// LS Electric XG5000 project: T7_ETH_485_20221121_AfterHeat-CYB60-BT-AP4
// PLC NewPLC
// module base 0 slot 1: 내장위치결정:XBF-PO02E (오픈컬렉터형, 2축)
// module base 0 slot 2: Cnet:XBL-C41A (Cnet 통신 모듈(RS-422/485))

PROGRAM 7k_pwm (task: 스캔 프로그램)

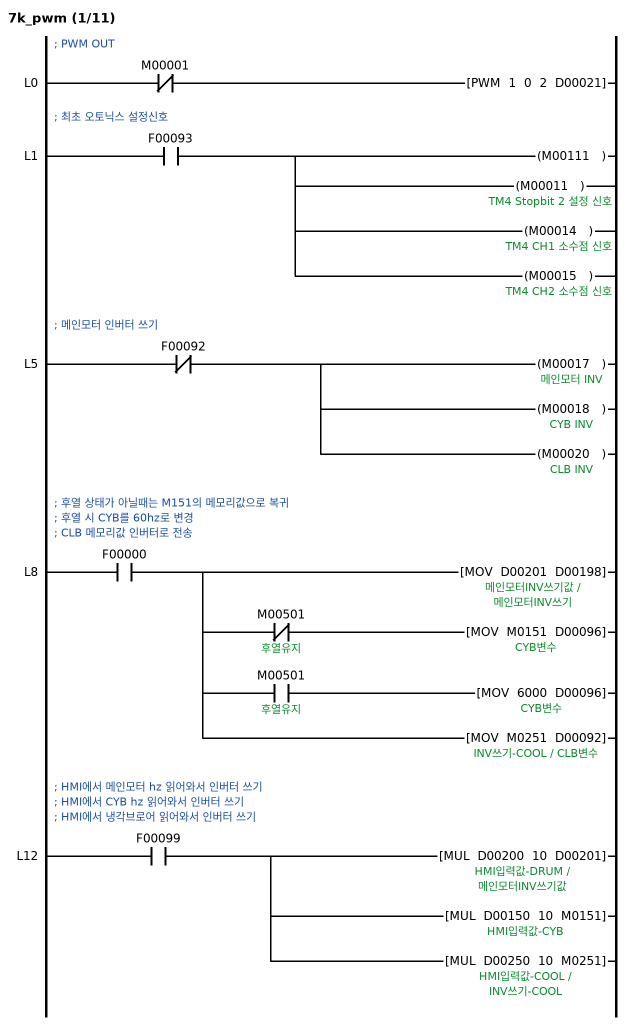
; L0
LOAD NOT  M00001
PWM       1 0 2 D00021
// output comment: PWM OUT
; L1
LOAD      F00093
OUT       M00111
OUT       M00011	// TM4 Stopbit 2 설정 신호
OUT       M00014	// TM4 CH1 소수점 신호
OUT       M00015	// TM4 CH2 소수점 신호
// output comment: 최초 오토닉스 설정신호
; L5
LOAD NOT  F00092
OUT       M00017	// 메인모터 INV
OUT       M00018	// CYB INV
OUT       M00020	// CLB INV
// output comment: 메인모터 인버터 쓰기
; L8
LOAD      F00000
MOV       D00201 D00198	// 메인모터INV쓰기값 / 메인모터INV쓰기
MPUSH
AND NOT   M00501	// 후열유지
MOV       M0151 D00096	// CYB변수
MLOAD
AND       M00501	// 후열유지
MOV       6000 D00096	// CYB변수
MPOP
MOV       M0251 D00092	// INV쓰기-COOL / CLB변수
// output comment: 후열 상태가 아닐때는 M151의 메모리값으로 복귀
// output comment: 후열 시 CYB를 60hz로 변경
// output comment: CLB 메모리값 인버터로 전송
; L12
LOAD      F00099
MUL       D00200 10 D00201	// HMI입력값-DRUM / 메인모터INV쓰기값
MUL       D00150 10 M0151	// HMI입력값-CYB
MUL       D00250 10 M0251	// HMI입력값-COOL / INV쓰기-COOL
// output comment: HMI에서 메인모터 hz 읽어와서 인버터 쓰기
// output comment: HMI에서 CYB hz 읽어와서 인버터 쓰기
// output comment: HMI에서 냉각브로어 읽어와서 인버터 쓰기

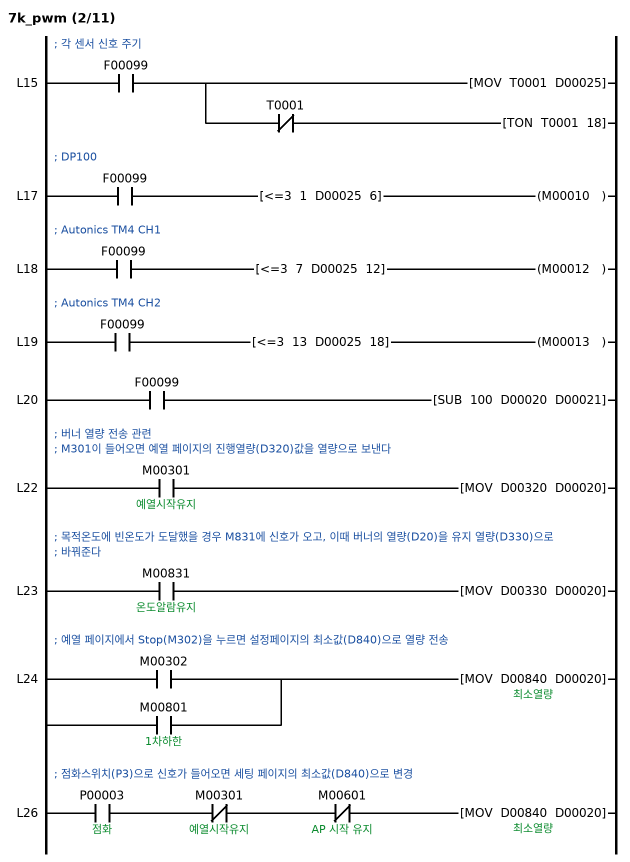
; L15
LOAD      F00099
MOV       T0001 D00025
AND NOT   T0001
TON       T0001 18
// output comment: 각 센서 신호 주기
; L17
LOAD      F00099
AND<=3    1 D00025 6
OUT       M00010
// output comment: DP100
; L18
LOAD      F00099
AND<=3    7 D00025 12
OUT       M00012
// output comment: Autonics TM4 CH1
; L19
LOAD      F00099
AND<=3    13 D00025 18
OUT       M00013
// output comment: Autonics TM4 CH2
; L20
LOAD      F00099
SUB       100 D00020 D00021
// 버너 열량 전송 관련
; L22
LOAD      M00301	// 예열시작유지
MOV       D00320 D00020
// output comment: M301이 들어오면 예열 페이지의 진행열량(D320)값을 열량으로 보낸다
; L23
LOAD      M00831	// 온도알람유지
MOV       D00330 D00020
// output comment: 목적온도에 빈온도가 도달했을 경우 M831에 신호가 오고, 이때 버너의 열량(D20)을 유지 열량(D330)으로 바꿔준다
; L24
LOAD      M00302
OR        M00801	// 1차하한
MOV       D00840 D00020	// 최소열량
// output comment: 예열 페이지에서 Stop(M302)을 누르면 설정페이지의 최소값(D840)으로 열량 전송
; L26
LOAD      P00003	// 점화
AND NOT   M00301	// 예열시작유지
AND NOT   M00601	// AP 시작 유지
MOV       D00840 D00020	// 최소열량
// output comment: 점화스위치(P3)으로 신호가 들어오면 세팅 페이지의 최소값(D840)으로 변경

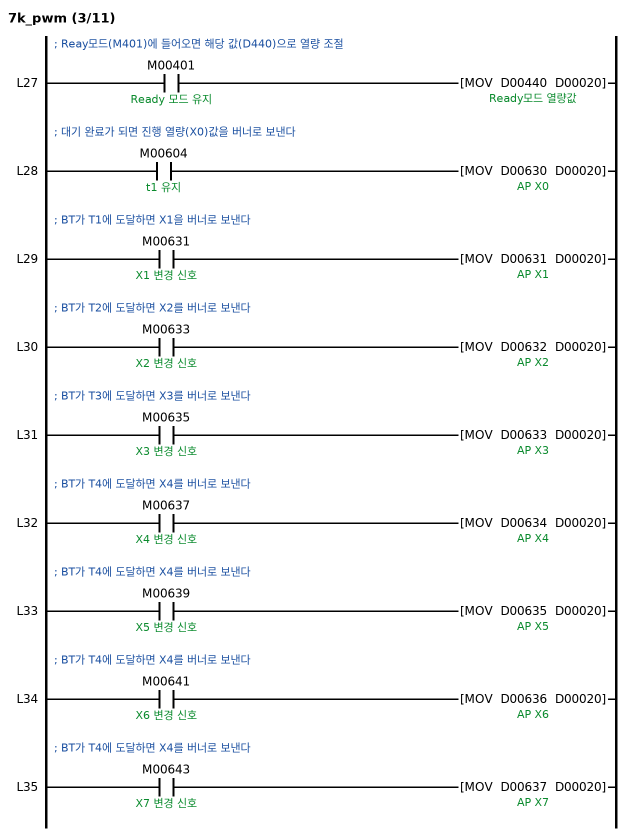
; L27
LOAD      M00401	// Ready 모드 유지
MOV       D00440 D00020	// Ready모드 열량값
// output comment: Reay모드(M401)에 들어오면 해당 값(D440)으로 열량 조절
; L28
LOAD      M00604	// t1 유지
MOV       D00630 D00020	// AP X0
// output comment: 대기 완료가 되면 진행 열량(X0)값을 버너로 보낸다
; L29
LOAD      M00631	// X1 변경 신호
MOV       D00631 D00020	// AP X1
// output comment: BT가 T1에 도달하면 X1을 버너로 보낸다
; L30
LOAD      M00633	// X2 변경 신호
MOV       D00632 D00020	// AP X2
// output comment: BT가 T2에 도달하면 X2를 버너로 보낸다
; L31
LOAD      M00635	// X3 변경 신호
MOV       D00633 D00020	// AP X3
// output comment: BT가 T3에 도달하면 X3를 버너로 보낸다
; L32
LOAD      M00637	// X4 변경 신호
MOV       D00634 D00020	// AP X4
// output comment: BT가 T4에 도달하면 X4를 버너로 보낸다
; L33
LOAD      M00639	// X5 변경 신호
MOV       D00635 D00020	// AP X5
// output comment: BT가 T4에 도달하면 X4를 버너로 보낸다
; L34
LOAD      M00641	// X6 변경 신호
MOV       D00636 D00020	// AP X6
// output comment: BT가 T4에 도달하면 X4를 버너로 보낸다
; L35
LOAD      M00643	// X7 변경 신호
MOV       D00637 D00020	// AP X7
// output comment: BT가 T4에 도달하면 X4를 버너로 보낸다

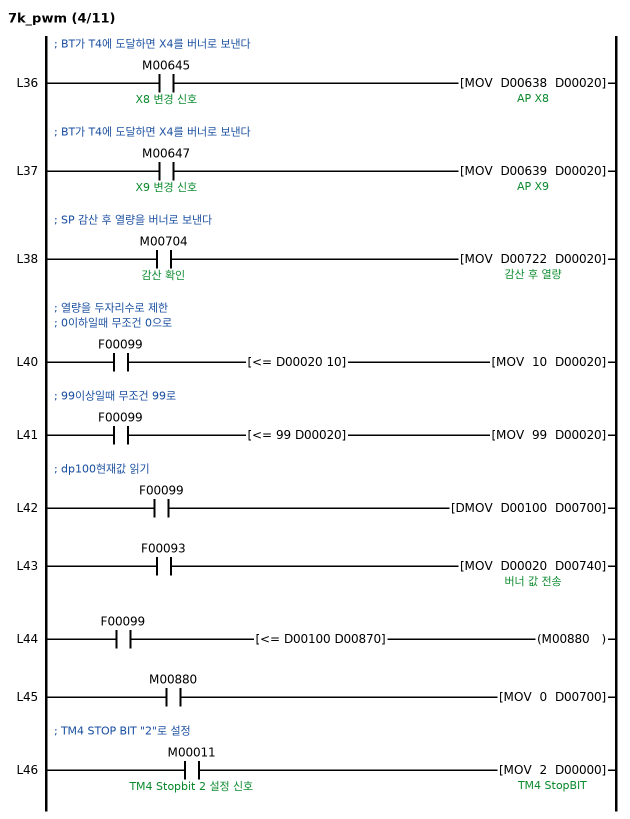
; L36
LOAD      M00645	// X8 변경 신호
MOV       D00638 D00020	// AP X8
// output comment: BT가 T4에 도달하면 X4를 버너로 보낸다
; L37
LOAD      M00647	// X9 변경 신호
MOV       D00639 D00020	// AP X9
// output comment: BT가 T4에 도달하면 X4를 버너로 보낸다
; L38
LOAD      M00704	// 감산 확인
MOV       D00722 D00020	// 감산 후 열량
// output comment: SP 감산 후 열량을 버너로 보낸다
// 열량을 두자리수로 제한
; L40
LOAD      F00099
AND<=     D00020 10
MOV       10 D00020
// output comment: 0이하일때 무조건 0으로
; L41
LOAD      F00099
AND<=     99 D00020
MOV       99 D00020
// output comment: 99이상일때 무조건 99로
; L42
LOAD      F00099
DMOV      D00100 D00700
// output comment: dp100현재값 읽기
; L43
LOAD      F00093
MOV       D00020 D00740	// 버너 값 전송
; L44
LOAD      F00099
AND<=     D00100 D00870
OUT       M00880
; L45
LOAD      M00880
MOV       0 D00700
; L46
LOAD      M00011	// TM4 Stopbit 2 설정 신호
MOV       2 D00000	// TM4 StopBIT
// output comment: TM4 STOP BIT "2"로 설정

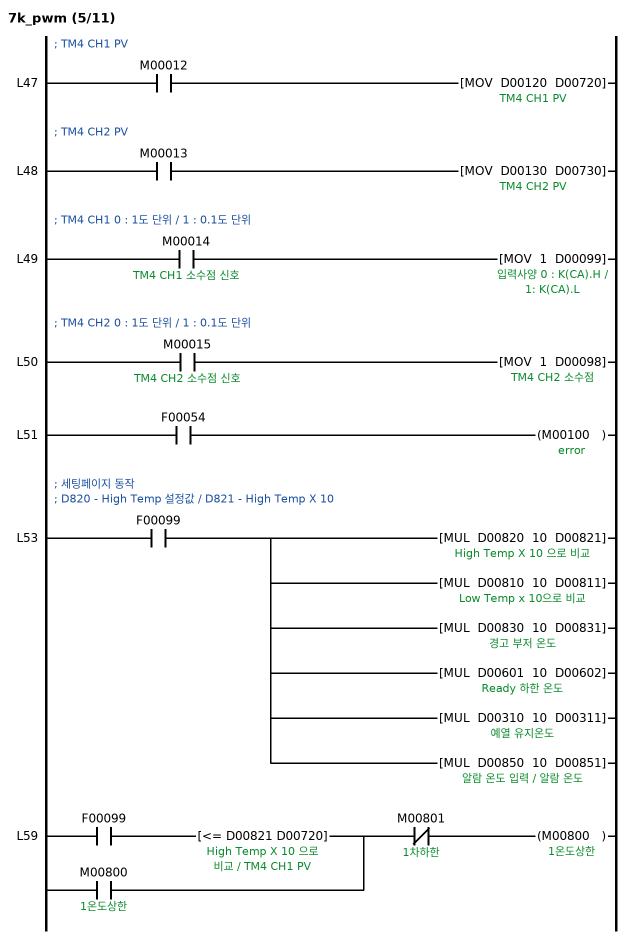
; L47
LOAD      M00012
MOV       D00120 D00720	// TM4 CH1 PV
// output comment: TM4 CH1 PV
; L48
LOAD      M00013
MOV       D00130 D00730	// TM4 CH2 PV
// output comment: TM4 CH2 PV
; L49
LOAD      M00014	// TM4 CH1 소수점 신호
MOV       1 D00099	// 입력사양 0 : K(CA).H / 1: K(CA).L
// output comment: TM4 CH1 0 : 1도 단위 / 1 : 0.1도 단위
; L50
LOAD      M00015	// TM4 CH2 소수점 신호
MOV       1 D00098	// TM4 CH2 소수점
// output comment: TM4 CH2 0 : 1도 단위 / 1 : 0.1도 단위
; L51
LOAD      F00054
OUT       M00100	// error
// 세팅페이지 동작
; L53
LOAD      F00099
MUL       D00820 10 D00821	// High Temp X 10 으로 비교
MUL       D00810 10 D00811	// Low Temp x 10으로 비교
MUL       D00830 10 D00831	// 경고 부저 온도
MUL       D00601 10 D00602	// Ready 하한 온도
MUL       D00310 10 D00311	// 예열 유지온도
MUL       D00850 10 D00851	// 알람 온도 입력 / 알람 온도 
// output comment: D820 - High Temp 설정값 / D821 - High Temp X 10
; L59
LOAD      F00099
AND<=     D00821 D00720	// High Temp X 10 으로 비교 / TM4 CH1 PV
OR        M00800	// 1온도상한
AND NOT   M00801	// 1차하한
OUT       M00800	// 1온도상한

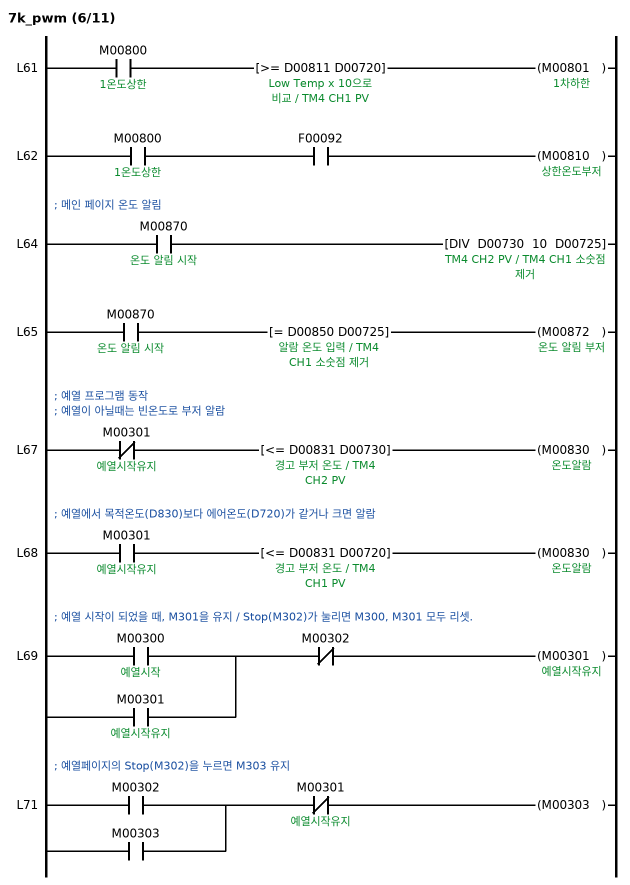
; L61
LOAD      M00800	// 1온도상한
AND>=     D00811 D00720	// Low Temp x 10으로 비교 / TM4 CH1 PV
OUT       M00801	// 1차하한
; L62
LOAD      M00800	// 1온도상한
AND       F00092
OUT       M00810	// 상한온도부저
// 메인 페이지 온도 알림
; L64
LOAD      M00870	// 온도 알림 시작
DIV       D00730 10 D00725	// TM4 CH2 PV / TM4 CH1 소숫점 제거
; L65
LOAD      M00870	// 온도 알림 시작
AND=      D00850 D00725	// 알람 온도 입력 / TM4 CH1 소숫점 제거
OUT       M00872	// 온도 알림 부저
// 예열 프로그램 동작
; L67
LOAD NOT  M00301	// 예열시작유지
AND<=     D00831 D00730	// 경고 부저 온도 / TM4 CH2 PV
OUT       M00830	// 온도알람
// output comment: 예열이 아닐때는 빈온도로 부저 알람
; L68
LOAD      M00301	// 예열시작유지
AND<=     D00831 D00720	// 경고 부저 온도 / TM4 CH1 PV
OUT       M00830	// 온도알람
// output comment: 예열에서 목적온도(D830)보다 에어온도(D720)가 같거나 크면 알람
; L69
LOAD      M00300	// 예열시작
OR        M00301	// 예열시작유지
AND NOT   M00302
OUT       M00301	// 예열시작유지
// output comment: 예열 시작이 되었을 때, M301을 유지 / Stop(M302)가 눌리면 M300, M301 모두 리셋.
; L71
LOAD      M00302
OR        M00303
AND NOT   M00301	// 예열시작유지
OUT       M00303
// output comment: 예열페이지의 Stop(M302)을 누르면 M303 유지

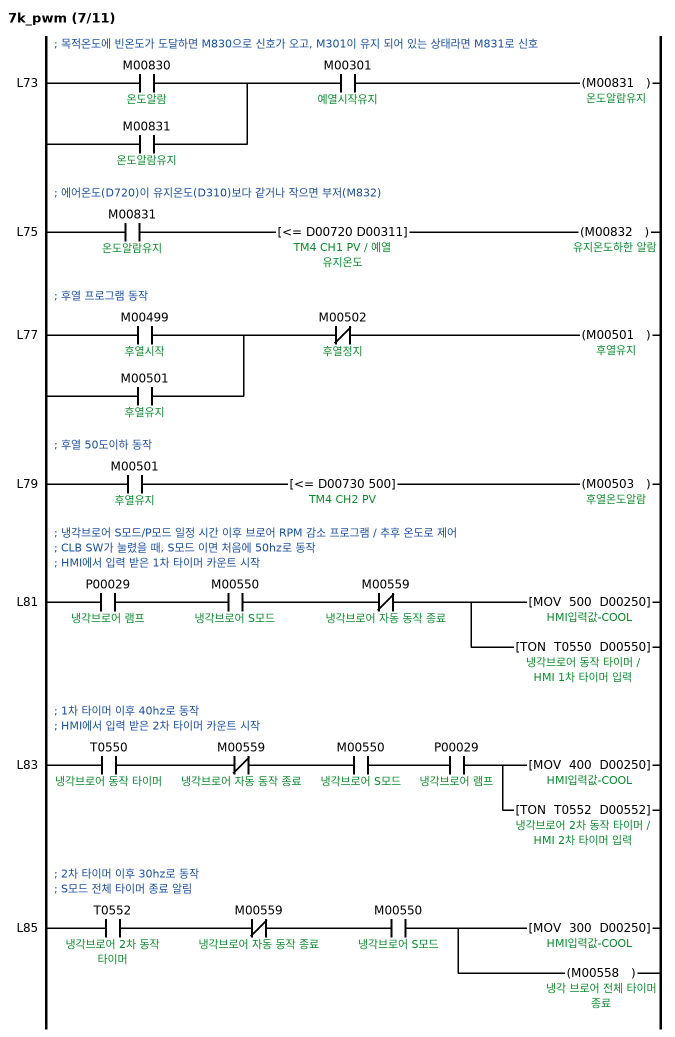
; L73
LOAD      M00830	// 온도알람
OR        M00831	// 온도알람유지
AND       M00301	// 예열시작유지
OUT       M00831	// 온도알람유지
// output comment: 목적온도에 빈온도가 도달하면 M830으로 신호가 오고, M301이 유지 되어 있는 상태라면 M831로 신호
; L75
LOAD      M00831	// 온도알람유지
AND<=     D00720 D00311	// TM4 CH1 PV / 예열 유지온도
OUT       M00832	// 유지온도하한 알람
// output comment: 에어온도(D720)이 유지온도(D310)보다 같거나 작으면 부저(M832)
// 후열 프로그램 동작
; L77
LOAD      M00499	// 후열시작
OR        M00501	// 후열유지
AND NOT   M00502	// 후열정지
OUT       M00501	// 후열유지
; L79
LOAD      M00501	// 후열유지
AND<=     D00730 500	// TM4 CH2 PV
OUT       M00503	// 후열온도알람
// output comment: 후열 50도이하 동작
// 냉각브로어 S모드/P모드 일정 시간 이후 브로어 RPM 감소 프로그램 / 추후 온도로 제어
; L81
LOAD      P00029	// 냉각브로어 램프
AND       M00550	// 냉각브로어 S모드
AND NOT   M00559	// 냉각브로어 자동 동작 종료
MOV       500 D00250	// HMI입력값-COOL
TON       T0550 D00550	// 냉각브로어 동작 타이머 / HMI 1차 타이머 입력
// output comment: CLB SW가 눌렸을 때, S모드 이면 처음에 50hz로 동작
// output comment: HMI에서 입력 받은 1차 타이머 카운트 시작
; L83
LOAD      T0550	// 냉각브로어 동작 타이머
AND NOT   M00559	// 냉각브로어 자동 동작 종료
AND       M00550	// 냉각브로어 S모드
AND       P00029	// 냉각브로어 램프
MOV       400 D00250	// HMI입력값-COOL
TON       T0552 D00552	// 냉각브로어 2차 동작 타이머 / HMI 2차 타이머 입력
// output comment: 1차 타이머 이후 40hz로 동작
// output comment: HMI에서 입력 받은 2차 타이머 카운트 시작
; L85
LOAD      T0552	// 냉각브로어 2차 동작 타이머
AND NOT   M00559	// 냉각브로어 자동 동작 종료
AND       M00550	// 냉각브로어 S모드
MOV       300 D00250	// HMI입력값-COOL
OUT       M00558	// 냉각 브로어 전체 타이머 종료
// output comment: 2차 타이머 이후 30hz로 동작
// output comment: S모드 전체 타이머 종료 알림

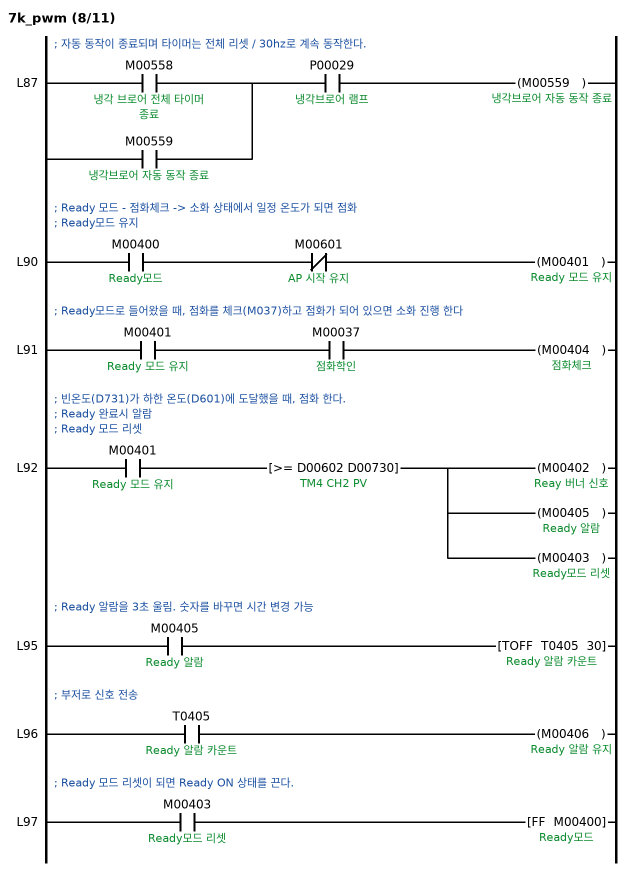
; L87
LOAD      M00558	// 냉각 브로어 전체 타이머 종료
OR        M00559	// 냉각브로어 자동 동작 종료
AND       P00029	// 냉각브로어 램프
OUT       M00559	// 냉각브로어 자동 동작 종료
// output comment: 자동 동작이 종료되며 타이머는 전체 리셋 / 30hz로 계속 동작한다.
// Ready 모드 - 점화체크 -> 소화 상태에서 일정 온도가 되면 점화
; L90
LOAD      M00400	// Ready모드
AND NOT   M00601	// AP 시작 유지
OUT       M00401	// Ready 모드 유지
// output comment: Ready모드 유지
; L91
LOAD      M00401	// Ready 모드 유지
AND       M00037	// 점화학인
OUT       M00404	// 점화체크
// output comment: Ready모드로 들어왔을 때, 점화를 체크(M037)하고 점화가 되어 있으면 소화 진행 한다
; L92
LOAD      M00401	// Ready 모드 유지
AND>=     D00602 D00730	// TM4 CH2 PV
OUT       M00402	// Reay 버너 신호
OUT       M00405	// Ready 알람
OUT       M00403	// Ready모드 리셋
// output comment: 빈온도(D731)가 하한 온도(D601)에 도달했을 때, 점화 한다.
// output comment: Ready 완료시 알람
// output comment: Ready 모드 리셋
; L95
LOAD      M00405	// Ready 알람
TOFF      T0405 30	// Ready 알람 카운트
// output comment: Ready 알람을 3초 울림. 숫자를 바꾸면 시간 변경 가능
; L96
LOAD      T0405	// Ready 알람 카운트
OUT       M00406	// Ready 알람 유지
// output comment: 부저로 신호 전송
; L97
LOAD      M00403	// Ready모드 리셋
FF        M00400	// Ready모드
// output comment: Ready 모드 리셋이 되면 Ready ON 상태를 끈다.

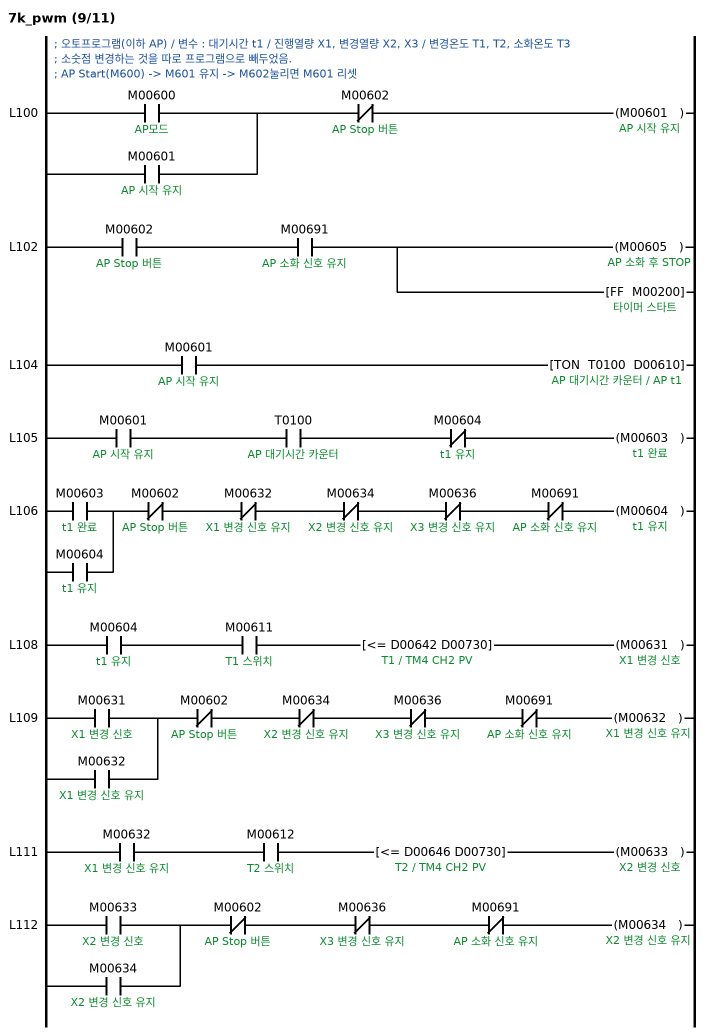
// 오토프로그램(이하 AP) / 변수 : 대기시간 t1 / 진행열량 X1, 변경열량 X2, X3 / 변경온도 T1, T2, 소화온도 T3
// 소숫점 변경하는 것을 따로 프로그램으로 빼두었음.
; L100
LOAD      M00600	// AP모드
OR        M00601	// AP 시작 유지
AND NOT   M00602	// AP Stop 버튼
OUT       M00601	// AP 시작 유지
// output comment: AP Start(M600) -> M601 유지 -> M602눌리면 M601 리셋
; L102
LOAD      M00602	// AP Stop 버튼
AND       M00691	// AP 소화 신호 유지
OUT       M00605	// AP 소화 후 STOP
FF        M00200	// 타이머 스타트
; L104
LOAD      M00601	// AP 시작 유지
TON       T0100 D00610	// AP 대기시간 카운터 / AP t1
; L105
LOAD      M00601	// AP 시작 유지
AND       T0100	// AP 대기시간 카운터
AND NOT   M00604	// t1 유지
OUT       M00603	// t1 완료
; L106
LOAD      M00603	// t1 완료
OR        M00604	// t1 유지
AND NOT   M00602	// AP Stop 버튼
AND NOT   M00632	// X1 변경 신호 유지
AND NOT   M00634	// X2 변경 신호 유지
AND NOT   M00636	// X3 변경 신호 유지
AND NOT   M00691	// AP 소화 신호 유지
OUT       M00604	// t1 유지
; L108
LOAD      M00604	// t1 유지
AND       M00611	// T1 스위치
AND<=     D00642 D00730	// T1 / TM4 CH2 PV
OUT       M00631	// X1 변경 신호
; L109
LOAD      M00631	// X1 변경 신호
OR        M00632	// X1 변경 신호 유지
AND NOT   M00602	// AP Stop 버튼
AND NOT   M00634	// X2 변경 신호 유지
AND NOT   M00636	// X3 변경 신호 유지
AND NOT   M00691	// AP 소화 신호 유지
OUT       M00632	// X1 변경 신호 유지
; L111
LOAD      M00632	// X1 변경 신호 유지
AND       M00612	// T2 스위치
AND<=     D00646 D00730	// T2 / TM4 CH2 PV
OUT       M00633	// X2 변경 신호
; L112
LOAD      M00633	// X2 변경 신호
OR        M00634	// X2 변경 신호 유지
AND NOT   M00602	// AP Stop 버튼
AND NOT   M00636	// X3 변경 신호 유지
AND NOT   M00691	// AP 소화 신호 유지
OUT       M00634	// X2 변경 신호 유지

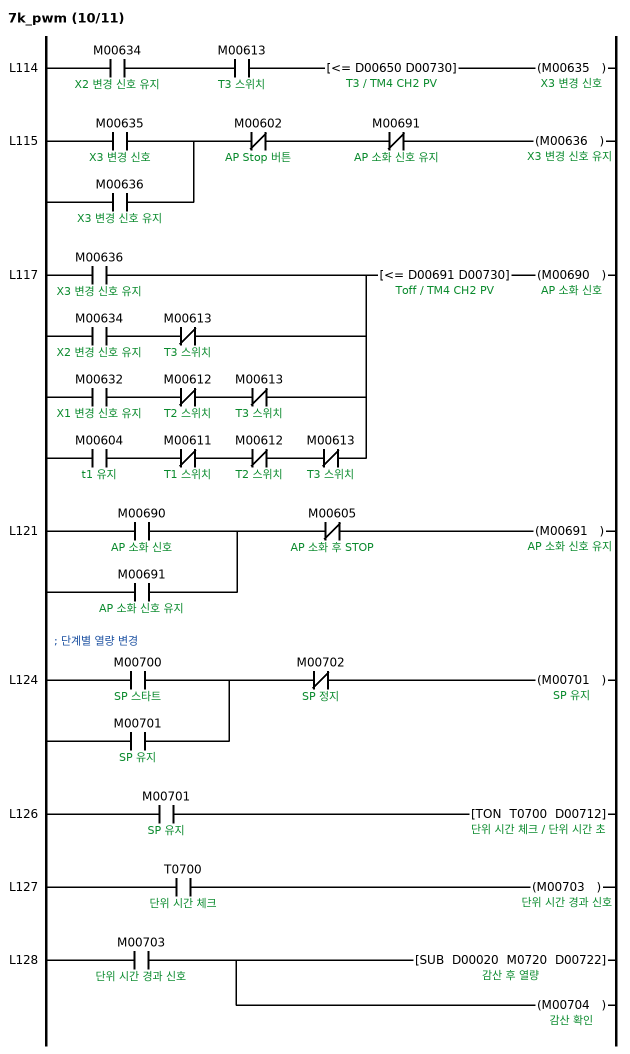
; L114
LOAD      M00634	// X2 변경 신호 유지
AND       M00613	// T3 스위치
AND<=     D00650 D00730	// T3 / TM4 CH2 PV
OUT       M00635	// X3 변경 신호
; L115
LOAD      M00635	// X3 변경 신호
OR        M00636	// X3 변경 신호 유지
AND NOT   M00602	// AP Stop 버튼
AND NOT   M00691	// AP 소화 신호 유지
OUT       M00636	// X3 변경 신호 유지
; L117
LOAD      M00636	// X3 변경 신호 유지
LOAD      M00634	// X2 변경 신호 유지
AND NOT   M00613	// T3 스위치
OR LOAD
LOAD      M00632	// X1 변경 신호 유지
AND NOT   M00612	// T2 스위치
AND NOT   M00613	// T3 스위치
OR LOAD
LOAD      M00604	// t1 유지
AND NOT   M00611	// T1 스위치
AND NOT   M00612	// T2 스위치
AND NOT   M00613	// T3 스위치
OR LOAD
AND<=     D00691 D00730	// Toff / TM4 CH2 PV
OUT       M00690	// AP 소화 신호
; L121
LOAD      M00690	// AP 소화 신호
OR        M00691	// AP 소화 신호 유지
AND NOT   M00605	// AP 소화 후 STOP
OUT       M00691	// AP 소화 신호 유지
// 단계별 열량 변경
; L124
LOAD      M00700	// SP 스타트
OR        M00701	// SP 유지
AND NOT   M00702	// SP 정지
OUT       M00701	// SP 유지
; L126
LOAD      M00701	// SP 유지
TON       T0700 D00712	// 단위 시간 체크 / 단위 시간 초
; L127
LOAD      T0700	// 단위 시간 체크
OUT       M00703	// 단위 시간 경과 신호
; L128
LOAD      M00703	// 단위 시간 경과 신호
SUB       D00020 M0720 D00722	// 감산 후 열량
OUT       M00704	// 감산 확인

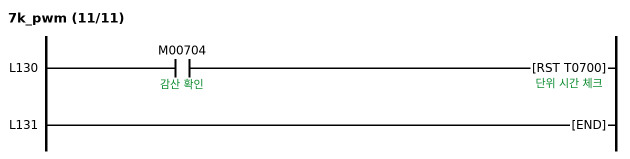
; L130
LOAD      M00704	// 감산 확인
RST       T0700	// 단위 시간 체크
; L131
END

PROGRAM 타이머 (task: 스캔 프로그램)

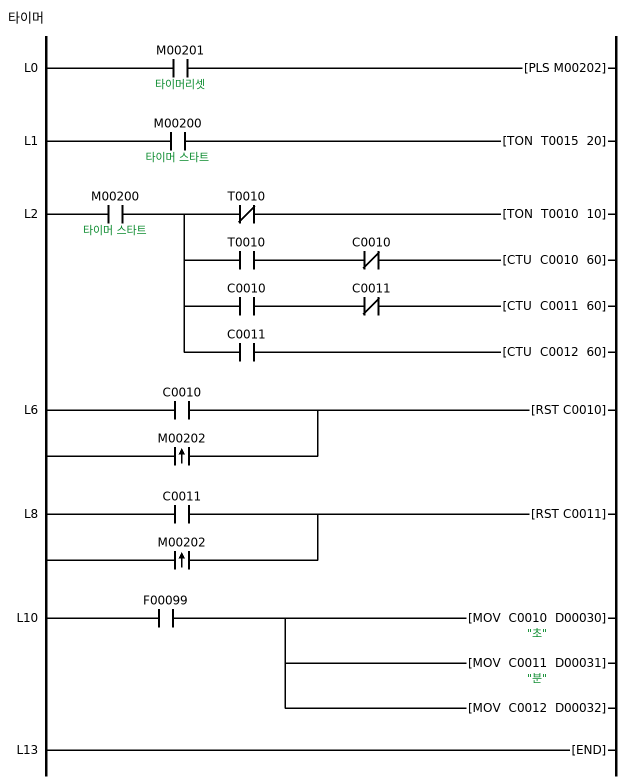
; L0
LOAD      M00201	// 타이머리셋
OUTP      M00202
; L1
LOAD      M00200	// 타이머 스타트
TON       T0015 20
; L2
LOAD      M00200	// 타이머 스타트
MPUSH
AND NOT   T0010
TON       T0010 10
MLOAD
AND       T0010
AND NOT   C0010
CTU       C0010 60
MLOAD
AND       C0010
AND NOT   C0011
CTU       C0011 60
MPOP
AND       C0011
CTU       C0012 60
; L6
LOAD      C0010
ORP       M00202
RST       C0010
; L8
LOAD      C0011
ORP       M00202
RST       C0011
; L10
LOAD      F00099
MOV       C0010 D00030	// "초"
MOV       C0011 D00031	// "분"
MOV       C0012 D00032
; L13
END

PROGRAM control (task: 스캔 프로그램)

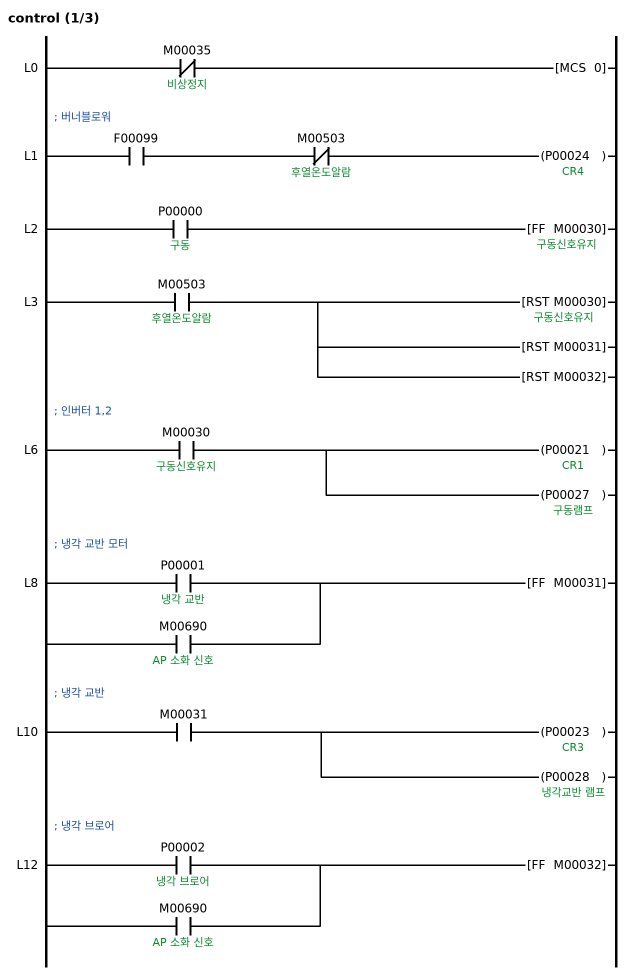
; L0
LOAD NOT  M00035	// 비상정지
MCS       0
; L1
LOAD      F00099
AND NOT   M00503	// 후열온도알람
OUT       P00024	// CR4
// output comment: 버너블로워
; L2
LOAD      P00000	// 구동
FF        M00030	// 구동신호유지
; L3
LOAD      M00503	// 후열온도알람
RST       M00030	// 구동신호유지
RST       M00031
RST       M00032
; L6
LOAD      M00030	// 구동신호유지
OUT       P00021	// CR1
OUT       P00027	// 구동램프
// output comment: 인버터 1,2
; L8
LOAD      P00001	// 냉각 교반
OR        M00690	// AP 소화 신호
FF        M00031
// output comment: 냉각 교반 모터
; L10
LOAD      M00031
OUT       P00023	// CR3
OUT       P00028	// 냉각교반 램프
// output comment: 냉각 교반
; L12
LOAD      P00002	// 냉각 브로어
OR        M00690	// AP 소화 신호
FF        M00032
// output comment: 냉각 브로어

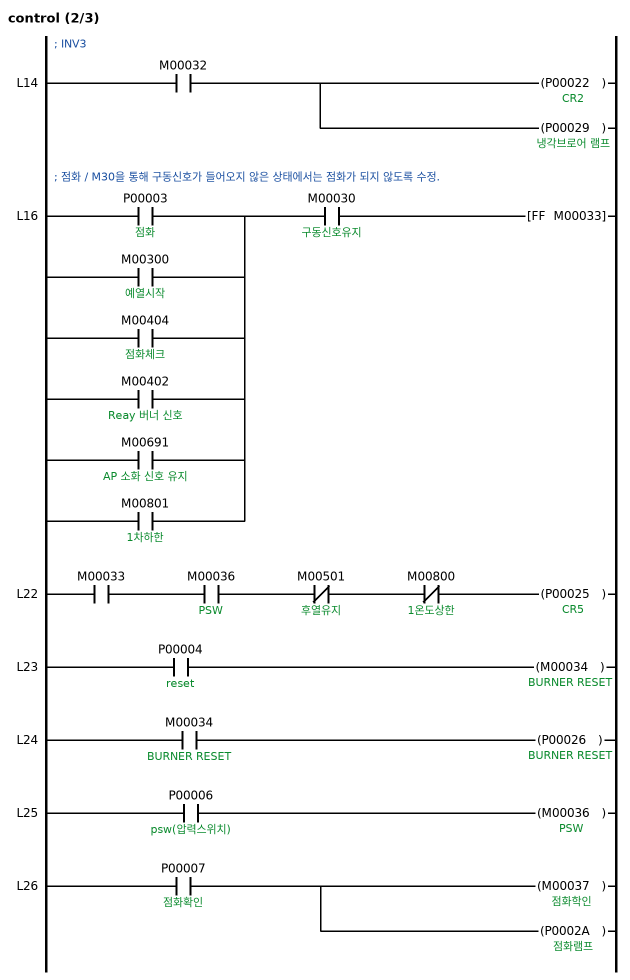
; L14
LOAD      M00032
OUT       P00022	// CR2
OUT       P00029	// 냉각브로어 램프
// output comment: INV3
; L16
LOAD      P00003	// 점화
OR        M00300	// 예열시작
OR        M00404	// 점화체크
OR        M00402	// Reay 버너 신호
OR        M00691	// AP 소화 신호 유지
OR        M00801	// 1차하한
AND       M00030	// 구동신호유지
FF        M00033
// output comment: 점화 / M30을 통해 구동신호가 들어오지 않은 상태에서는 점화가 되지 않도록 수정.
; L22
LOAD      M00033
AND       M00036	// PSW
AND NOT   M00501	// 후열유지
AND NOT   M00800	// 1온도상한
OUT       P00025	// CR5
; L23
LOAD      P00004	// reset
OUT       M00034	// BURNER RESET
; L24
LOAD      M00034	// BURNER RESET
OUT       P00026	// BURNER RESET
; L25
LOAD      P00006	// psw(압력스위치)
OUT       M00036	// PSW
; L26
LOAD      P00007	// 점화확인
OUT       M00037	// 점화학인
OUT       P0002A	// 점화램프

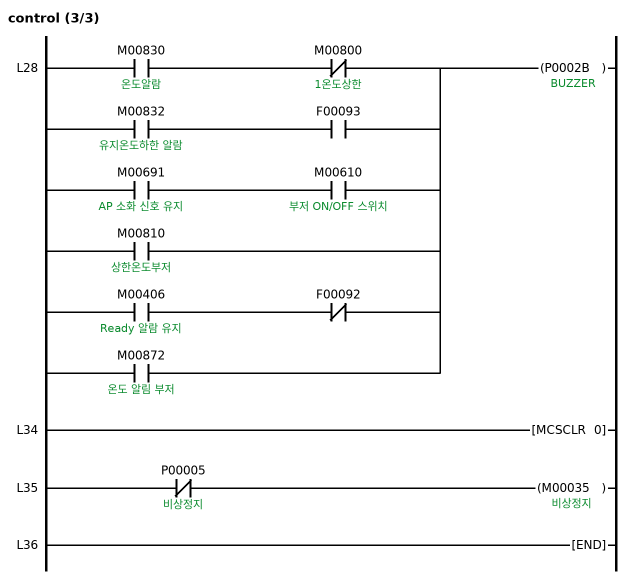
; L28
LOAD      M00830	// 온도알람
AND NOT   M00800	// 1온도상한
LOAD      M00832	// 유지온도하한 알람
AND       F00093
OR LOAD
LOAD      M00691	// AP 소화 신호 유지
AND       M00610	// 부저 ON/OFF 스위치
OR LOAD
OR        M00810	// 상한온도부저
LOAD      M00406	// Ready 알람 유지
AND NOT   F00092
OR LOAD
OR        M00872	// 온도 알림 부저
OUT       P0002B	// BUZZER
; L34
MCSCLR    0
; L35
LOAD NOT  P00005	// 비상정지
OUT       M00035	// 비상정지
; L36
END

PROGRAM 소숫점_변경 (task: 스캔 프로그램)

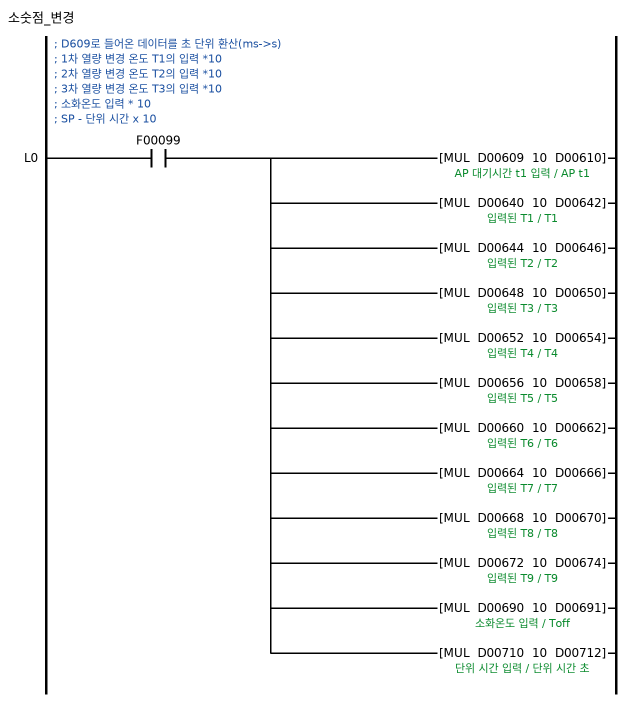
; L0
LOAD      F00099
MUL       D00609 10 D00610	// AP 대기시간 t1 입력 / AP t1
MUL       D00640 10 D00642	// 입력된 T1 / T1
MUL       D00644 10 D00646	// 입력된 T2 / T2
MUL       D00648 10 D00650	// 입력된 T3 / T3
MUL       D00652 10 D00654	// 입력된 T4 / T4
MUL       D00656 10 D00658	// 입력된 T5 / T5
MUL       D00660 10 D00662	// 입력된 T6 / T6
MUL       D00664 10 D00666	// 입력된 T7 / T7
MUL       D00668 10 D00670	// 입력된 T8 / T8
MUL       D00672 10 D00674	// 입력된 T9 / T9
MUL       D00690 10 D00691	// 소화온도 입력 / Toff
MUL       D00710 10 D00712	// 단위 시간 입력 / 단위 시간 초
// output comment: D609로 들어온 데이터를 초 단위 환산(ms->s)
// output comment: 1차 열량 변경 온도 T1의 입력 *10
// output comment: 2차 열량 변경 온도 T2의 입력 *10
// output comment: 3차 열량 변경 온도 T3의 입력 *10
// output comment: 소화온도 입력 * 10
// output comment: SP - 단위 시간 x 10

PROGRAM 예열_후열_타이머 (task: 스캔 프로그램)

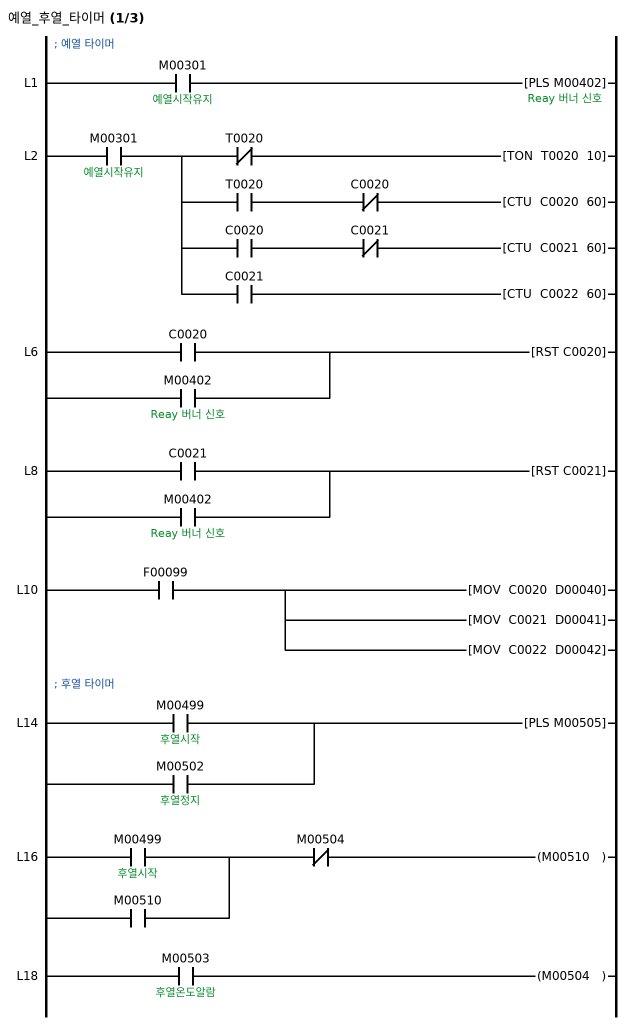
// 예열 타이머
; L1
LOAD      M00301	// 예열시작유지
OUTP      M00402	// Reay 버너 신호
; L2
LOAD      M00301	// 예열시작유지
MPUSH
AND NOT   T0020
TON       T0020 10
MLOAD
AND       T0020
AND NOT   C0020
CTU       C0020 60
MLOAD
AND       C0020
AND NOT   C0021
CTU       C0021 60
MPOP
AND       C0021
CTU       C0022 60
; L6
LOAD      C0020
OR        M00402	// Reay 버너 신호
RST       C0020
; L8
LOAD      C0021
OR        M00402	// Reay 버너 신호
RST       C0021
; L10
LOAD      F00099
MOV       C0020 D00040
MOV       C0021 D00041
MOV       C0022 D00042
// 후열 타이머
; L14
LOAD      M00499	// 후열시작
OR        M00502	// 후열정지
OUTP      M00505
; L16
LOAD      M00499	// 후열시작
OR        M00510
AND NOT   M00504
OUT       M00510
; L18
LOAD      M00503	// 후열온도알람
OUT       M00504

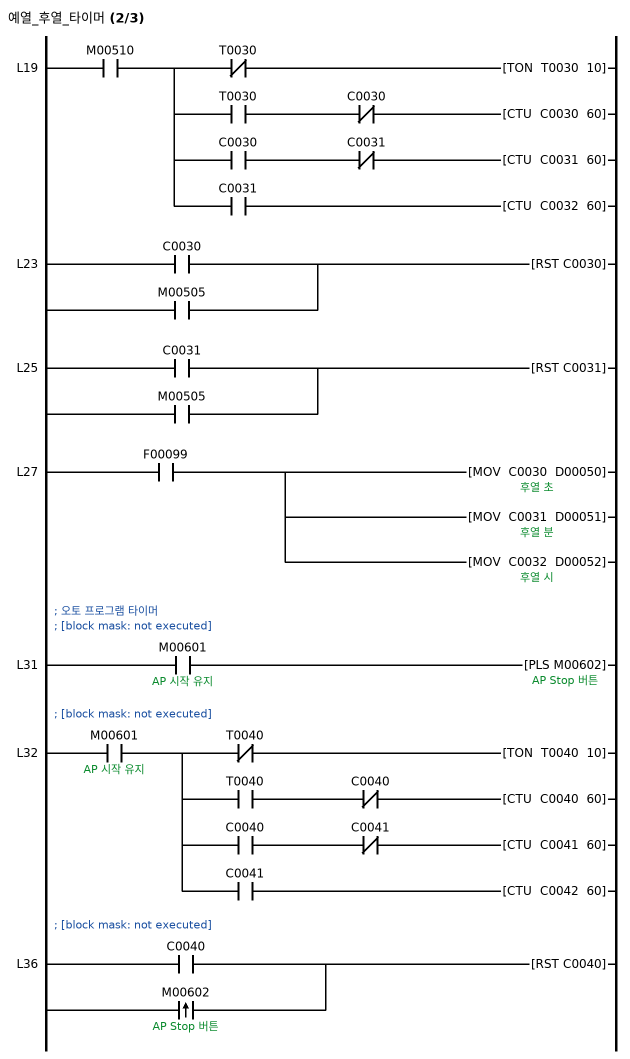
; L19
LOAD      M00510
MPUSH
AND NOT   T0030
TON       T0030 10
MLOAD
AND       T0030
AND NOT   C0030
CTU       C0030 60
MLOAD
AND       C0030
AND NOT   C0031
CTU       C0031 60
MPOP
AND       C0031
CTU       C0032 60
; L23
LOAD      C0030
OR        M00505
RST       C0030
; L25
LOAD      C0031
OR        M00505
RST       C0031
; L27
LOAD      F00099
MOV       C0030 D00050	// 후열 초
MOV       C0031 D00051	// 후열 분
MOV       C0032 D00052	// 후열 시
// 오토 프로그램 타이머
; L31 (block mask: not executed)
LOAD      M00601	// AP 시작 유지
OUTP      M00602	// AP Stop 버튼
; L32 (block mask: not executed)
LOAD      M00601	// AP 시작 유지
MPUSH
AND NOT   T0040
TON       T0040 10
MLOAD
AND       T0040
AND NOT   C0040
CTU       C0040 60
MLOAD
AND       C0040
AND NOT   C0041
CTU       C0041 60
MPOP
AND       C0041
CTU       C0042 60
; L36 (block mask: not executed)
LOAD      C0040
ORP       M00602	// AP Stop 버튼
RST       C0040

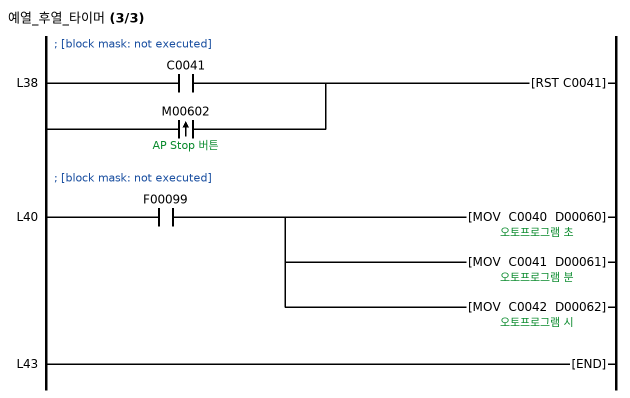
; L38 (block mask: not executed)
LOAD      C0041
ORP       M00602	// AP Stop 버튼
RST       C0041
; L40 (block mask: not executed)
LOAD      F00099
MOV       C0040 D00060	// 오토프로그램 초
MOV       C0041 D00061	// 오토프로그램 분
MOV       C0042 D00062	// 오토프로그램 시
; L43
END

PROGRAM 485_ARTISAN (task: 스캔 프로그램)

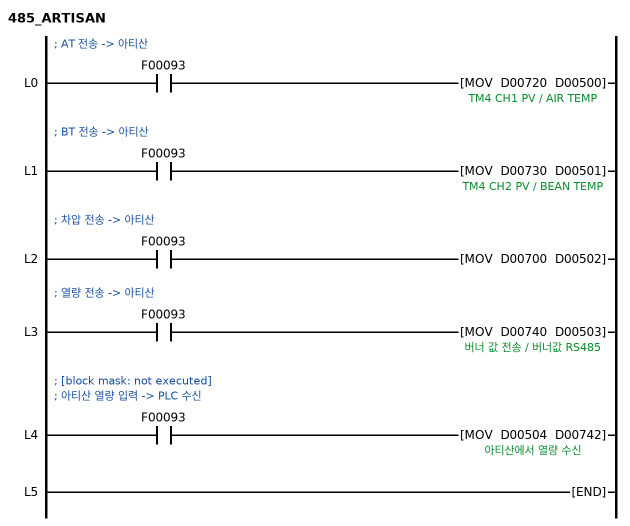
; L0
LOAD      F00093
MOV       D00720 D00500	// TM4 CH1 PV / AIR TEMP
// output comment: AT 전송 -> 아티산
; L1
LOAD      F00093
MOV       D00730 D00501	// TM4 CH2 PV / BEAN TEMP
// output comment: BT 전송 -> 아티산
; L2
LOAD      F00093
MOV       D00700 D00502
// output comment: 차압 전송 -> 아티산
; L3
LOAD      F00093
MOV       D00740 D00503	// 버너 값 전송 / 버너값 RS485
// output comment: 열량 전송 -> 아티산
; L4 (block mask: not executed)
LOAD      F00093
MOV       D00504 D00742	// 아티산에서 열량 수신
// output comment: 아티산 열량 입력 -> PLC 수신
; L5
END

VARIABLES AND COMMENTS (devices not used above)
P00020	BIT	BURNER PWM
D00930	WORD	1차 조절 온도
D00620	WORD	TM4 CH1 PV : 소수점없음
D00600	WORD	Ready Temp
M00016	BIT	인버터 CYB
D00199	WORD	1번인버터읽기
D00197	WORD	CYB INV 쓰기
D00202	WORD	CYB INV 쓰기값
D00203	WORD	HMI CYB INV 설정값
M00019	BIT	CYB INV 신호
D00196	WORD	CYB INV 읽기
D00204	WORD	INV 쓰기
M0710	WORD	단위 시간 입력
M0722	WORD	감산 후 열량
D01609	WORD	t1 레시피1
D01610	WORD	AP t1
D01630	WORD	X1 레시피1
D01631	WORD	X2 레시피1
D01632	WORD	X3 레시피1
D01633	WORD	X4 레시피1
D01640	WORD	T1 레시피1
D01644	WORD	T2 레시피1
D01648	WORD	T3 레시피1
D01690	WORD	소화온도 레시피1
D02609	WORD	t1 레시피2
D02630	WORD	X1 레시피2
D02631	WORD	X2 레시피2
D02632	WORD	X3 레시피2
D02633	WORD	X4 레시피2
D02640	WORD	T1 레시피2
D02644	WORD	T2 레시피2
D02648	WORD	T3 레시피2
D02690	WORD	소화온도 레시피2
D03609	WORD	t1 레시피3
D03630	WORD	X1 레시피3
D03631	WORD	X2 레시피3
D03632	WORD	X3 레시피3
D03633	WORD	X4 레시피3
D03640	WORD	T1 레시피3
D03644	WORD	T2 레시피3
D03648	WORD	T3 레시피3
D03690	WORD	소화온도 레시피3
D04609	WORD	t1 레시피4
D04630	WORD	X1 레시피4
D04631	WORD	X2 레시피4
D04632	WORD	X3 레시피4
D04633	WORD	X4 레시피4
D04640	WORD	T1 레시피4
D04644	WORD	T2 레시피4
D04648	WORD	T3 레시피4
D04690	WORD	소화온도 레시피4
D05609	WORD	t1 레시피5
D05630	WORD	X1 레시피5
D05631	WORD	X2 레시피5
D05632	WORD	X3 레시피5
D05633	WORD	X4 레시피5
D05640	WORD	T1 레시피5
D05644	WORD	T2 레시피5
D05648	WORD	T3 레시피5
D05690	WORD	소화온도 레시피5
D06609	WORD	t1 레시피6
D06630	WORD	X1 레시피6
D06631	WORD	X2 레시피6
D06632	WORD	X3 레시피6
D06633	WORD	X4 레시피6
D06640	WORD	T1 레시피6
D06644	WORD	T2 레시피6
D06648	WORD	T3 레시피6
D06690	WORD	소화온도 레시피6
D07609	WORD	t1 레시피7
D07630	WORD	X1 레시피7
D07631	WORD	X2 레시피7
D07632	WORD	X3 레시피7
D07633	WORD	X4 레시피7
D07640	WORD	T1 레시피7
D07644	WORD	T2 레시피7
D07648	WORD	T3 레시피7
D07690	WORD	소화온도 레시피7
D08609	WORD	t1 레시피8
D08630	WORD	X1 레시피8
D08631	WORD	X2 레시피8
D08632	WORD	X3 레시피8
D08633	WORD	X4 레시피8
D08640	WORD	T1 레시피8
D08644	WORD	T2 레시피8
D08648	WORD	T3 레시피8
D08690	WORD	소화온도 레시피8
D09609	WORD	t1 레시피9
D09630	WORD	X1 레시피9
D09631	WORD	X2 레시피9
D09632	WORD	X3 레시피9
D09633	WORD	X4 레시피9
D09640	WORD	T1 레시피9
D09644	WORD	T2 레시피9
D09648	WORD	T3 레시피9
D09690	WORD	소화온도 레시피9
D10609	WORD	t1 레시피10
D10630	WORD	X1 레시피10
D10631	WORD	X2 레시피10
D10632	WORD	X3 레시피10
D10633	WORD	X4 레시피10
D10640	WORD	T1 레시피10
D10644	WORD	T2 레시피10
D10648	WORD	T3 레시피10
D10690	WORD	소화온도 레시피10
D11609	WORD	t1 레시피11
D11630	WORD	X1 레시피11
D11631	WORD	X2 레시피11
D11632	WORD	X3 레시피11
D11633	WORD	X4 레시피11
D11640	WORD	T1 레시피11
D11644	WORD	T2 레시피11
D11648	WORD	T3 레시피11
D11690	WORD	소화온도 레시피11
D12609	WORD	t1 레시피12
D12630	WORD	X1 레시피12
D12631	WORD	X2 레시피12
D12632	WORD	X3 레시피12
D12633	WORD	X4 레시피12
D12640	WORD	T1 레시피12
D12644	WORD	T2 레시피12
D12648	WORD	T3 레시피12
D12690	WORD	소화온도 레시피12
D13609	WORD	t1 레시피13
D13630	WORD	X1 레시피13
D13631	WORD	X2 레시피13
D13632	WORD	X3 레시피13
D13633	WORD	X4 레시피13
D13640	WORD	T1 레시피13
D13644	WORD	T2 레시피13
D13648	WORD	T3 레시피13
D13690	WORD	소화온도 레시피13
D14609	WORD	t1 레시피14
D14630	WORD	X1 레시피14
D14631	WORD	X2 레시피14
D14632	WORD	X3 레시피14
D14633	WORD	X4 레시피14
D14640	WORD	T1 레시피14
D14644	WORD	T2 레시피14
D14648	WORD	T3 레시피14
D14690	WORD	소화온도 레시피14
D15609	WORD	t1 레시피15
D15630	WORD	X1 레시피15
D15631	WORD	X2 레시피15
D15632	WORD	X3 레시피15
D15633	WORD	X4 레시피15
D15640	WORD	T1 레시피15
D15644	WORD	T2 레시피15
D15648	WORD	T3 레시피15
D15690	WORD	소화온도 레시피15
D16609	WORD	t1 레시피16
D16630	WORD	X1 레시피16
D16631	WORD	X2 레시피16
D16632	WORD	X3 레시피16
D16633	WORD	X4 레시피16
D16640	WORD	T1 레시피16
D16644	WORD	T2 레시피16
D16648	WORD	T3 레시피16
D16690	WORD	소화온도 레시피16
M00850	BIT	온도 알림 시작
M00852	BIT	온도 알림 부저
M00873	BIT	부저 유지
D00748	WORD	아티산 체크
M00552	BIT	55Hz 동작 종료
M00638	BIT	X4 변경 신호 유지
M00630	BIT	t1 유지 체크
M00640	BIT	X5 변경 신호 유지
M00642	BIT	X6 변경 신호 유지
M00644	BIT	X7 변경 신호 유지
M00646	BIT	X8 변경 신호 유지
M00648	BIT	X9 변경 신호 유지
M00614	BIT	T4 스위치
M00615	BIT	T5 스위치
M00616	BIT	T6 스위치
M00617	BIT	T7 스위치
M00618	BIT	T8 스위치
M00619	BIT	T9 스위치